TYPE ICCD : 
STRUCT
	bComOpen:BOOL;  //扫码Tcp 开
    bComClose:BOOL;  //扫码Tcp 关

	bSend :BOOL; //  扫码开
	//bLOFF :BOOL; //扫码关
	bDone  :BOOL; //扫码完成
    bError :BOOL;//扫码故障	
    strReceive:STRING;//

END_STRUCT
END_TYPE

(* stored: Version 1.1.0.1, ProductVersion 3.1.4024.9
   DUT ICCD: Id {52f5e6ff-faf3-4530-9e72-5fec59e4e18d} *)
